Universal Robots PolyScope program: Pour_coffee.urp

Program Pour_coffee (installation=default directory=/programs/DMS createdIn=5.8.2.10297 lastSavedIn=5.12.6.1102099 robotSerialNumber=20215500597)
Calibrated DH parameters: a=[0.000193, -0.066673, -0.391568, -0.000012, 0.00005, 0]; d=[0.162643, -472.05677, 465.132521, 7.058239, 0.099746, 0.099582]; alpha=[1.571116, 0.00089, 0.003862, 1.569269, -1.569248, 0]; deltaTheta=[0, -1.413394, 7.628392, 0.068187, 0, -0.000001]
Robot Program (runOnlyOnce=true)
  num_loop := 5
  looped := 0
  URCap Gripper Activate (Robotiq_Grippers, Robotiq Inc.) dataModel(ResetAndActivateKey=false)
  URCap Gripper (Robotiq_Grippers, Robotiq Inc.) dataModel(position=81.25490196078431, force=100.0, speed=64.0, positionInDouble=81.25490196078431, forceInDouble=100.0, speedInDouble=64.0, slaveIds=[9], blocking=true)
  MoveJ speed 60 deg/s, acceleration 80 deg/s^2 (useActiveTCP=true) feature=Base
    Waypoint center1: TCP in base x=-78.565 y=-626.961 z=386.259 mm, rx=0.0116 ry=-2.2034 rz=2.2303 rad; joints [53.979, -98.506, 113.327, -15.86, 53.983, 180.13] deg; TCP offset x=0 y=0 z=191.5 mm, rx=0 ry=0 rz=0 rad
  center_2 := center1
  SuppressedNode
    MoveJ speed 60 deg/s, acceleration 80 deg/s^2 (useActiveTCP=true) feature=Base
      Waypoint pouring_1: TCP in base x=-78.85 y=-695.523 z=386.207 mm, rx=0.0145 ry=-2.8725 rz=1.2641 rad; joints [64.733, -68.042, 53.837, 59.508, 71.416, 161.757] deg
  pouring := pouring_1
  'Now Cotton Candy Creation'
  radius := 0.029
  SuppressedNode
    radius := 0.135
  height := 0
  SuppressedNode
    cold_start_wait := 101.25
  wait_time := 10
  pour_time_1 := 3.75
  SuppressedNode
    circle_time := GP_int_in[2]
  SuppressedNode
    wait_time := 1
  SuppressedNode
    pour_time := 33.75
  circle_time := 3.75
  SuppressedNode
    cold_start_spin := 28
  SuppressedNode
    cold_start_spin := 100
  SuppressedNode
    center := Joint_6_name
  center := pouring
  bottom := pose_add(center, p[0, -radius, height, 0, 0, 0])
  right := pose_add(center, p[-radius, 0, -height, 0, 0, 0])
  top_circ := pose_add(center, p[0, radius, height, 0, 0, 0])
  left := pose_add(center, p[radius, 0, -height, 0, 0, 0])
  SuppressedNode
    diff := pose_sub(left,bottom )
  SuppressedNode
    Loop While (checkContinuously=false) expression=circles_no>0
      MoveP speed 250 mm/s, acceleration 1200 mm/s^2 (blendRadius=0.125 useActiveTCP=true) feature=Base
        Waypoint Waypoint (Variable): variable=bottom
        CircleMove (OrientationMode=UNCONSTRAINED)
          Waypoint Waypoint (Variable): variable=left
          Waypoint Waypoint (Variable): variable(name=top_circ)
      MoveP speed 250 mm/s, acceleration 1200 mm/s^2 (blendRadius=0.025 useActiveTCP=true) feature=Base
        Waypoint Waypoint (Variable): variable=top_circ
        CircleMove (OrientationMode=UNCONSTRAINED)
          Waypoint Waypoint (Variable): variable(name=right)
          Waypoint Waypoint (Variable): variable=bottom
      circles_no := circles_no-1
  SuppressedNode
    Timer (action=Stop) variable(name=timer_3)
  SuppressedNode
    Wait Sleep waitTime=101.25
  SuppressedNode
    Wait Condition expression=GP_int_in[0]
  SuppressedNode
    Script: sleep(wait_time)
  SuppressedNode
    Timer (action=Start) variable(name=timer_1)
  Loop While (checkContinuously=false) expression=num_loop>looped
    pour_time := pour_time_1
    MoveP speed 200 mm/s, acceleration 1200 mm/s^2 (blendRadius=0.025 useActiveTCP=true) feature=Base
      Waypoint pouring_1 referenceName=pouring_1: motionParameters(jointSpeed=1.047198 jointAcceleration=1.396263 cartesianSpeed=0.06 cartesianAcceleration=0.9); TCP in base x=-75.666 y=-686.85 z=386.054 mm, rx=0.0145 ry=-2.8728 rz=1.2637 rad; joints [64.63, -69.536, 55.955, 58.928, 71.344, 161.678] deg
    Loop While (checkContinuously=false) expression=pour_time>0
      MoveP speed 56 mm/s, acceleration 1200 mm/s^2 (blendRadius=0.025 useActiveTCP=true) feature=Base
        Waypoint Waypoint (Variable): variable=bottom
        CircleMove (OrientationMode=UNCONSTRAINED)
          Waypoint Waypoint (Variable): variable=left
          Waypoint Waypoint (Variable): variable=top_circ
      MoveP speed 56 mm/s, acceleration 1200 mm/s^2 (blendRadius=0.025 useActiveTCP=true) feature=Base
        Waypoint Waypoint (Variable): variable=top_circ
        CircleMove (OrientationMode=UNCONSTRAINED)
          Waypoint Waypoint (Variable): variable=right
          Waypoint Waypoint (Variable): variable=bottom
      pour_time := pour_time-circle_time
    SuppressedNode
      MoveJ speed 60 deg/s, acceleration 80 deg/s^2 (useActiveTCP=true) feature=Base
        Waypoint pouring_1: TCP in base x=-75.697 y=-697.555 z=386.148 mm, rx=0.0144 ry=-2.8727 rz=1.2639 rad; joints [65.188, -67.798, 53.476, 59.528, 71.735, 162.095] deg
        Waypoint center1: TCP in base x=-78.565 y=-626.961 z=386.259 mm, rx=0.0116 ry=-2.2034 rz=2.2303 rad; joints [53.979, -98.506, 113.327, -15.86, 53.983, 180.13] deg
    SuppressedNode
      MoveP speed 56 mm/s, acceleration 1200 mm/s^2 (blendRadius=0.025 useActiveTCP=true) feature=Base
        Waypoint Waypoint (Variable): variable=bottom
        CircleMove (OrientationMode=UNCONSTRAINED)
          Waypoint Waypoint (Variable): variable=left
          Waypoint Waypoint (Variable): motionParameters(jointSpeed=1.047198 jointAcceleration=1.396263 cartesianSpeed=0.07 cartesianAcceleration=0.9); variable(name=center_2)
    MoveP speed 56 mm/s, acceleration 1200 mm/s^2 (blendRadius=0.025 useActiveTCP=true) feature=Base
      Waypoint Waypoint (Variable): variable=bottom
      CircleMove (OrientationMode=UNCONSTRAINED)
        Waypoint Waypoint (Variable): variable(name=pouring)
        Waypoint Waypoint (Variable): motionParameters(jointSpeed=1.047198 jointAcceleration=1.396263 cartesianSpeed=0.07 cartesianAcceleration=0.9); variable=center_2
    Script: looped = looped + 1
    Script: sleep(wait_time)
  MoveJ speed 60 deg/s, acceleration 80 deg/s^2 (useActiveTCP=true) feature=Base
    Waypoint center1: TCP in base x=-78.565 y=-626.961 z=386.259 mm, rx=0.0116 ry=-2.2034 rz=2.2303 rad; joints [53.979, -98.506, 113.327, -15.86, 53.983, 180.13] deg
  SuppressedNode
    Loop While (checkContinuously=false) expression=pour_time>0
      MoveP speed 56 mm/s, acceleration 1200 mm/s^2 (blendRadius=0.025 useActiveTCP=true) feature=Base
        Waypoint Waypoint (Variable): variable=bottom
        CircleMove (OrientationMode=UNCONSTRAINED)
          Waypoint Waypoint (Variable): variable=left
          Waypoint Waypoint (Variable): variable=top_circ
      MoveP speed 56 mm/s, acceleration 1200 mm/s^2 (blendRadius=0.025 useActiveTCP=true) feature=Base
        Waypoint Waypoint (Variable): variable=top_circ
        CircleMove (OrientationMode=UNCONSTRAINED)
          Waypoint Waypoint (Variable): variable=right
          Waypoint Waypoint (Variable): variable=bottom
      pour_time := pour_time-circle_time
  SuppressedNode
    MoveJ speed 60 deg/s, acceleration 80 deg/s^2 (useActiveTCP=true) feature=Base
      Waypoint Waypoint_2: TCP in base x=-24.03 y=651.793 z=574.352 mm, rx=-0.9882 ry=-1.0644 rz=-1.2372 rad; joints [248.909, -99.854, 96.502, -11.42, 64.977, 96.89] deg
      Waypoint Waypoint_5: TCP in base x=-65.345 y=508.583 z=589.478 mm, rx=-0.8529 ry=-1.3704 rz=-1.3892 rad; joints [239.18, -119.542, 101.662, 8.745, 51.039, 78.082] deg
      Waypoint Waypoint_12: TCP in base x=-341.731 y=349.139 z=446.744 mm, rx=1.0197 ry=-1.4327 rz=-1.9509 rad; joints [261.046, -128.059, 128.66, -21.395, 27.658, 2.719] deg
      Waypoint Waypoint_13: TCP in base x=-346.288 y=487.83 z=199.367 mm, rx=1.1258 ry=-1.8238 rz=-1.9724 rad; joints [274.508, -89.471, 132.703, -38.479, 53.378, -24.773] deg
      Waypoint base_position: TCP in base x=-328.73 y=482.036 z=140.622 mm, rx=1.1107 ry=-1.8448 rz=-1.9801 rad; joints [271.637, -83.004, 138.617, -50.548, 51.741, -25.068] deg
      URCap Gripper Activate (Robotiq_Grippers, Robotiq Inc.) dataModel(ResetAndActivateKey=false)
      URCap Gripper (Robotiq_Grippers, Robotiq Inc.) dataModel(position=0.0, force=0.0, speed=100.0, positionInDouble=0.0, forceInDouble=0.0, speedInDouble=100.0, slaveIds=[9], blocking=true)
      Waypoint Waypoint_14: TCP in base x=-273.276 y=422.463 z=166.295 mm, rx=0.9524 ry=-2.167 rz=-1.9141 rad; joints [271.624, -104.005, 143.852, -26.72, 64.174, -25.036] deg
      URCap Gripper (Robotiq_Grippers, Robotiq Inc.) dataModel(position=100.0, force=0.0, speed=100.0, positionInDouble=100.0, forceInDouble=0.0, speedInDouble=100.0, slaveIds=[9], blocking=true)
      Waypoint Waypoint_15: TCP in base x=-47.378 y=367.135 z=156.328 mm, rx=-1.8568 ry=-1.4579 rz=-0.9844 rad; joints [256.209, -119.497, 138.801, 14.851, 90.035, 90] deg; TCP offset x=0 y=0 z=191.5 mm, rx=0 ry=0 rz=0 rad
